TYPE st_PressureTransducer_Input :
STRUCT
	value : LREAL;
END_STRUCT
END_TYPE

(* stored: Version 1.1.0.1, ProductVersion 3.1.4024.9
   DUT st_PressureTransducer_Input: Id {1936f3f3-5f6b-428a-822b-5c57bbef157b} *)
